TYPE ST_EL3443_DPM_MUX_ULINT :
STRUCT
    nSelector : UINT := E_EL3443_DPM_Phase.Error_INDEX_Not_Valid;
    nValueRef : POINTER TO ULINT;
END_STRUCT
END_TYPE

(* stored: Version 1.1.0.1, ProductVersion 3.1.4024.4
   DUT ST_EL3443_DPM_MUX_ULINT: Id {e97de12d-9ae3-4ec0-8384-9bfeca34798d} *)
